// Mitsubishi GX Works2 project: 240423_우선동작순차회로   PLC: Q03UDV

PROGRAM MAIN
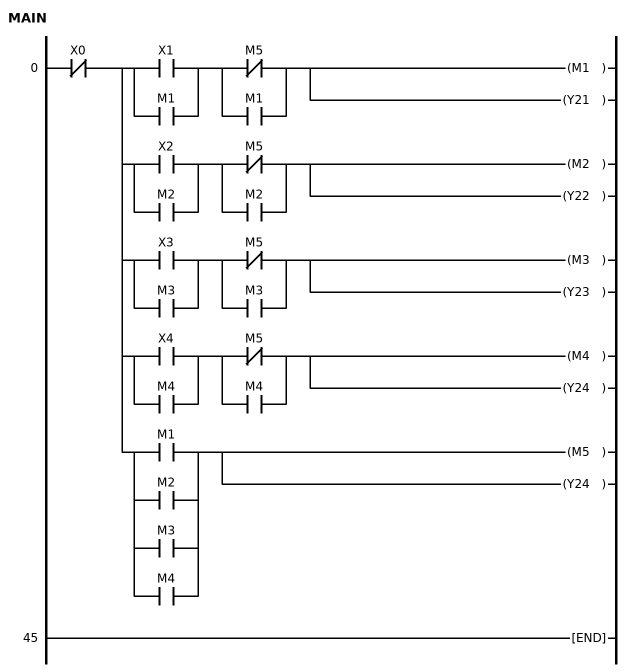
0     LDI     X0
      MPS
      LD      X1
      OR      M1
      ANB
      LDI     M5
      OR      M1
      ANB
      OUT     M1
      OUT     Y21
      MRD
      LD      X2
      OR      M2
      ANB
      LDI     M5
      OR      M2
      ANB
      OUT     M2
      OUT     Y22
      MRD
      LD      X3
      OR      M3
      ANB
      LDI     M5
      OR      M3
      ANB
      OUT     M3
      OUT     Y23
      MRD
      LD      X4
      OR      M4
      ANB
      LDI     M5
      OR      M4
      ANB
      OUT     M4
      OUT     Y24
      MPP
      LD      M1
      OR      M2
      OR      M3
      OR      M4
      ANB
      OUT     M5
      OUT     Y24
45    END
END_PROGRAM
